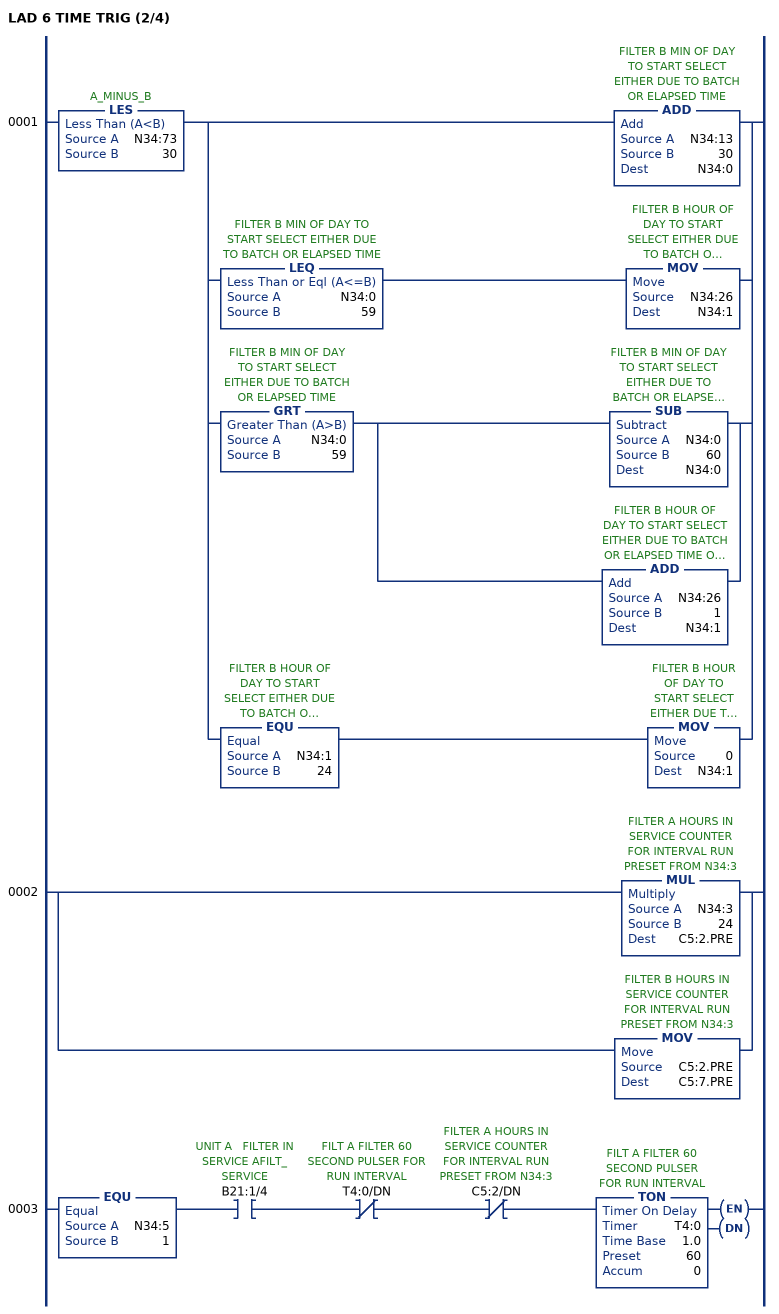
% Rung: 1 %
SOR LES N34:73 30 BST ADD N34:13 30 N34:0 NXB LEQ N34:0 59 MOV N34:26 N34:1 NXB GRT N34:0 59 BST SUB N34:0 60 N34:0 NXB ADD N34:26 1 N34:1 BND NXB EQU N34:1 24 MOV 0 N34:1 BND EOR
%   N34:73  A_MINUS_B %
%   N34:13  "FILTER A MIN OF DAY TO START SELECT EITHER DUE TO BATCH OR ELAPSED TIME" %
%   N34:0  "FILTER B MIN OF DAY TO START SELECT EITHER DUE TO BATCH OR ELAPSED TIME" %
%   N34:26  "FILTER A HOUR OF DAY TO START SELECT EITHER DUE TO BATCH OR ELAPSED TIME OR DP" %
%   N34:1  "FILTER B HOUR OF DAY TO START SELECT EITHER DUE TO BATCH OR ELAPSED TIME OR DP" %
% Rung: 2 %
SOR BST MUL N34:3 24 C5:2.PRE NXB MOV C5:2.PRE C5:7.PRE BND EOR
%   N34:3  "FILT INTERVAL IN DAYS TO START A REGN" %
%   C5:2  "FILTER A HOURS IN SERVICE COUNTER FOR INTERVAL RUN PRESET FROM N34:3" %
%   C5:7  "FILTER B HOURS IN SERVICE COUNTER FOR INTERVAL RUN PRESET FROM N34:3" %
% Rung: 3 %
SOR EQU N34:5 1 XIC B21:1/4 XIO T4:0/DN XIO C5:2/DN TON T4:0 1.0 60 0 EOR
%   B21:1/4  AFILT_SERVICE  "UNIT A   FILTER IN SERVICE" %
%   T4:0  "FILT A FILTER 60 SECOND PULSER FOR RUN INTERVAL" %
%   C5:2  "FILTER A HOURS IN SERVICE COUNTER FOR INTERVAL RUN PRESET FROM N34:3" %

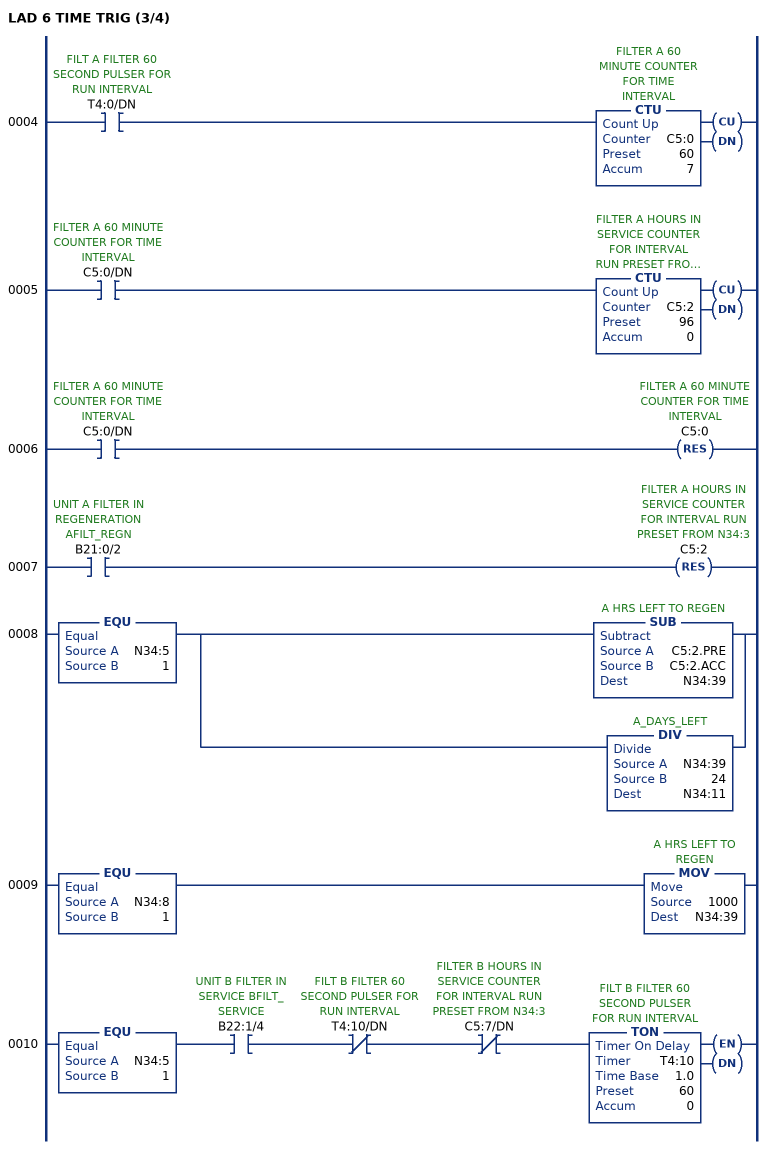
% Rung: 4 %
SOR XIC T4:0/DN CTU C5:0 60 7 EOR
%   T4:0  "FILT A FILTER 60 SECOND PULSER FOR RUN INTERVAL" %
%   C5:0  "FILTER A 60 MINUTE COUNTER FOR TIME INTERVAL" %
% Rung: 5 %
SOR XIC C5:0/DN CTU C5:2 96 0 EOR
%   C5:0  "FILTER A 60 MINUTE COUNTER FOR TIME INTERVAL" %
%   C5:2  "FILTER A HOURS IN SERVICE COUNTER FOR INTERVAL RUN PRESET FROM N34:3" %
% Rung: 6 %
SOR XIC C5:0/DN RES C5:0 EOR
%   C5:0  "FILTER A 60 MINUTE COUNTER FOR TIME INTERVAL" %
% Rung: 7 %
SOR XIC B21:0/2 RES C5:2 EOR
%   B21:0/2  AFILT_REGN  "UNIT A FILTER IN REGENERATION" %
%   C5:2  "FILTER A HOURS IN SERVICE COUNTER FOR INTERVAL RUN PRESET FROM N34:3" %
% Rung: 8 %
SOR EQU N34:5 1 BST SUB C5:2.PRE C5:2.ACC N34:39 NXB DIV N34:39 24 N34:11 BND EOR
%   C5:2  "FILTER A HOURS IN SERVICE COUNTER FOR INTERVAL RUN PRESET FROM N34:3" %
%   N34:39  "A HRS LEFT TO REGEN" %
%   N34:11  A_DAYS_LEFT %
% Rung: 9 %
SOR EQU N34:8 1 MOV 1000 N34:39 EOR
%   N34:39  "A HRS LEFT TO REGEN" %
% Rung: 10 %
SOR EQU N34:5 1 XIC B22:1/4 XIO T4:10/DN XIO C5:7/DN TON T4:10 1.0 60 0 EOR
%   B22:1/4  BFILT_SERVICE  "UNIT B FILTER IN SERVICE" %
%   T4:10  "FILT B FILTER 60 SECOND PULSER FOR RUN INTERVAL" %
%   C5:7  "FILTER B HOURS IN SERVICE COUNTER FOR INTERVAL RUN PRESET FROM N34:3" %

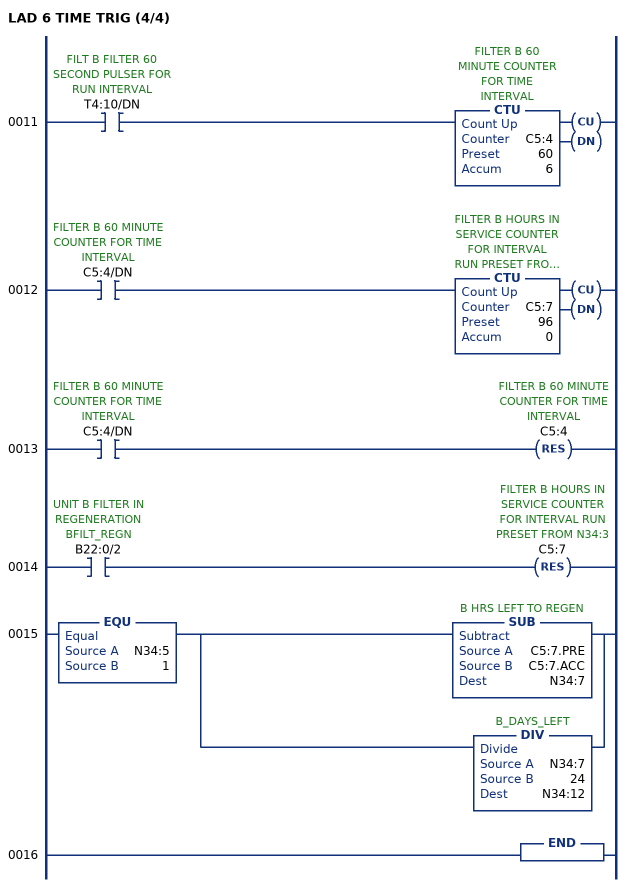
% Rung: 11 %
SOR XIC T4:10/DN CTU C5:4 60 6 EOR
%   T4:10  "FILT B FILTER 60 SECOND PULSER FOR RUN INTERVAL" %
%   C5:4  "FILTER B 60 MINUTE COUNTER FOR TIME INTERVAL" %
% Rung: 12 %
SOR XIC C5:4/DN CTU C5:7 96 0 EOR
%   C5:4  "FILTER B 60 MINUTE COUNTER FOR TIME INTERVAL" %
%   C5:7  "FILTER B HOURS IN SERVICE COUNTER FOR INTERVAL RUN PRESET FROM N34:3" %
% Rung: 13 %
SOR XIC C5:4/DN RES C5:4 EOR
%   C5:4  "FILTER B 60 MINUTE COUNTER FOR TIME INTERVAL" %
% Rung: 14 %
SOR XIC B22:0/2 RES C5:7 EOR
%   B22:0/2  BFILT_REGN  "UNIT B FILTER IN REGENERATION" %
%   C5:7  "FILTER B HOURS IN SERVICE COUNTER FOR INTERVAL RUN PRESET FROM N34:3" %
% Rung: 15 %
SOR EQU N34:5 1 BST SUB C5:7.PRE C5:7.ACC N34:7 NXB DIV N34:7 24 N34:12 BND EOR
%   C5:7  "FILTER B HOURS IN SERVICE COUNTER FOR INTERVAL RUN PRESET FROM N34:3" %
%   N34:7  "B HRS LEFT TO REGEN" %
%   N34:12  B_DAYS_LEFT %
% Rung: 16 %
SOR END EOR

LADDER 7 "A VESSEL"
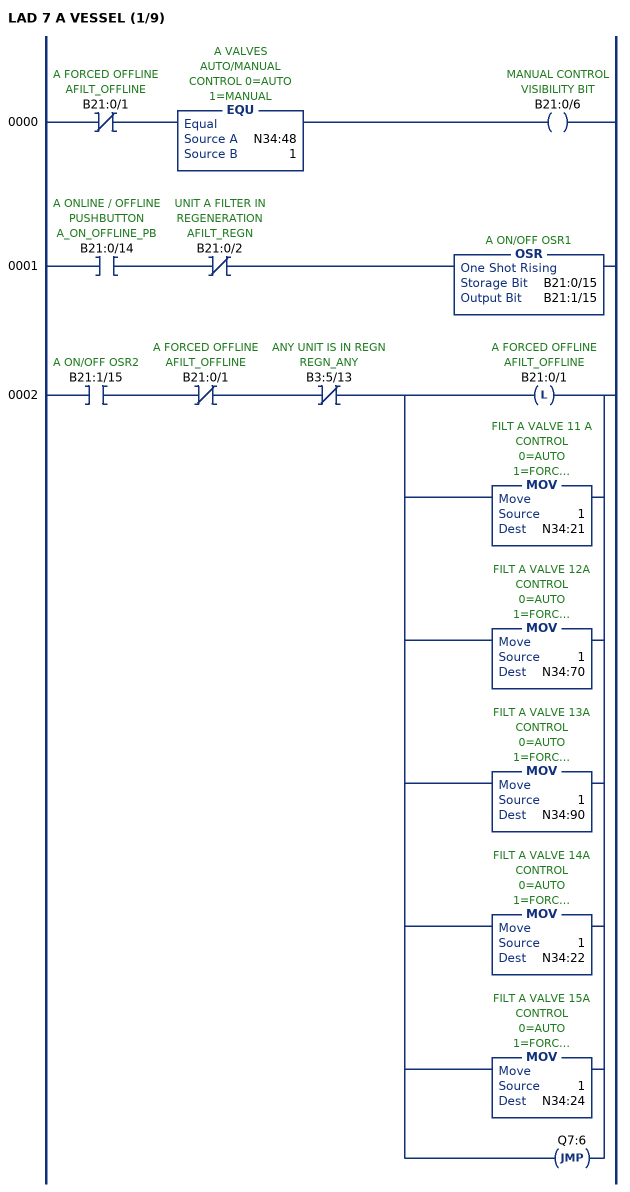
% Rung: 0 %
SOR XIO B21:0/1 EQU N34:48 1 OTE B21:0/6 EOR
%   B21:0/1  AFILT_OFFLINE  "A FORCED OFFLINE" %
%   N34:48  "A VALVES AUTO/MANUAL CONTROL 0=AUTO 1=MANUAL" %
%   B21:0/6  "MANUAL CONTROL VISIBILITY BIT" %
% Rung: 1 %
SOR XIC B21:0/14 XIO B21:0/2 OSR B21:0/15 B21:1/15 EOR
%   B21:0/14  A_ON_OFFLINE_PB  "A ONLINE / OFFLINE PUSHBUTTON" %
%   B21:0/2  AFILT_REGN  "UNIT A FILTER IN REGENERATION" %
%   B21:0/15  "A ON/OFF OSR1" %
%   B21:1/15  "A ON/OFF OSR2" %
% Rung: 2 %
SOR XIC B21:1/15 XIO B21:0/1 XIO B3:5/13 BST OTL B21:0/1 NXB MOV 1 N34:21 NXB MOV 1 N34:70 NXB MOV 1 N34:90 NXB MOV 1 N34:22 NXB MOV 1 N34:24 NXB JMP Q7:6 BND EOR
%   B21:1/15  "A ON/OFF OSR2" %
%   B21:0/1  AFILT_OFFLINE  "A FORCED OFFLINE" %
%   B3:5/13  REGN_ANY  "ANY UNIT IS IN REGN" %
%   N34:21  "FILT A VALVE 11 A CONTROL 0=AUTO 1=FORCE CLOSED 2=FORCE ON" %
%   N34:70  "FILT A VALVE 12A CONTROL 0=AUTO 1=FORCE CLOSED 2=FORCE ON" %
%   N34:90  "FILT A VALVE 13A CONTROL 0=AUTO 1=FORCE CLOSED 2=FORCE ON" %
%   N34:22  "FILT A VALVE 14A CONTROL 0=AUTO 1=FORCE CLOSED 2=FORCE ON" %
%   N34:24  "FILT A VALVE 15A CONTROL 0=AUTO 1=FORCE CLOSED 2=FORCE ON" %

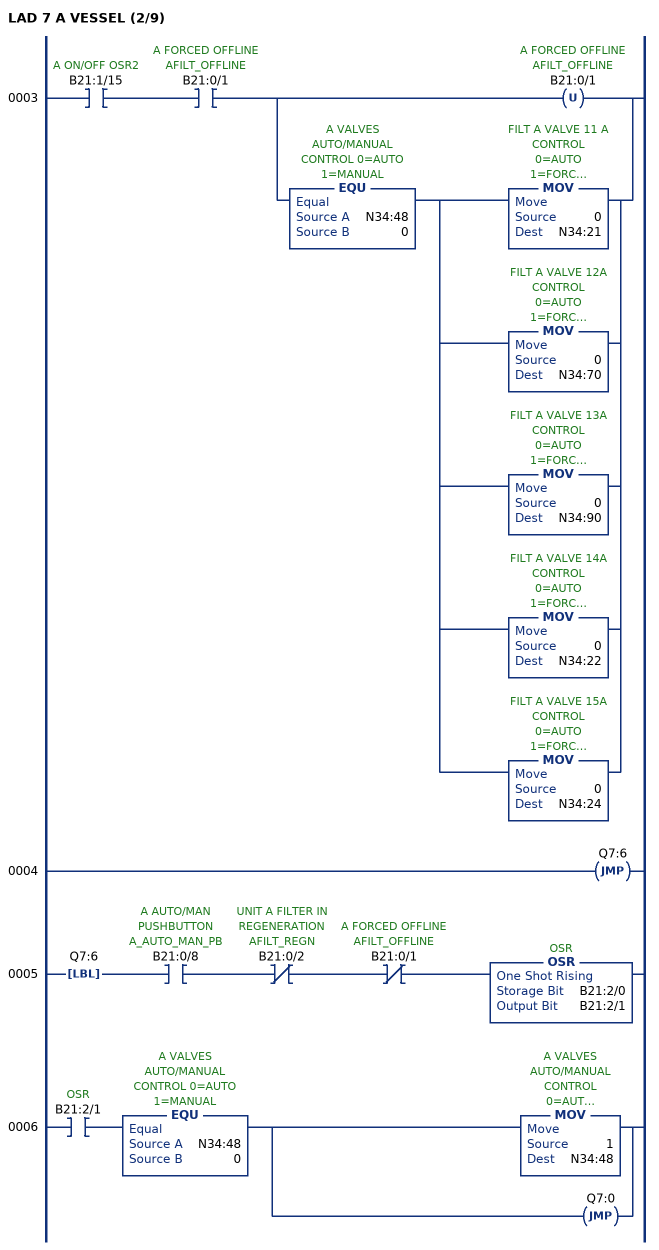
% Rung: 3 %
SOR XIC B21:1/15 XIC B21:0/1 BST OTU B21:0/1 NXB EQU N34:48 0 BST MOV 0 N34:21 NXB MOV 0 N34:70 NXB MOV 0 N34:90 NXB MOV 0 N34:22 NXB MOV 0 N34:24 BND BND EOR
%   B21:1/15  "A ON/OFF OSR2" %
%   B21:0/1  AFILT_OFFLINE  "A FORCED OFFLINE" %
%   N34:48  "A VALVES AUTO/MANUAL CONTROL 0=AUTO 1=MANUAL" %
%   N34:21  "FILT A VALVE 11 A CONTROL 0=AUTO 1=FORCE CLOSED 2=FORCE ON" %
%   N34:70  "FILT A VALVE 12A CONTROL 0=AUTO 1=FORCE CLOSED 2=FORCE ON" %
%   N34:90  "FILT A VALVE 13A CONTROL 0=AUTO 1=FORCE CLOSED 2=FORCE ON" %
%   N34:22  "FILT A VALVE 14A CONTROL 0=AUTO 1=FORCE CLOSED 2=FORCE ON" %
%   N34:24  "FILT A VALVE 15A CONTROL 0=AUTO 1=FORCE CLOSED 2=FORCE ON" %
% Rung: 4 %
SOR JMP Q7:6 EOR
% Rung: 5 %
SOR LBL Q7:6 XIC B21:0/8 XIO B21:0/2 XIO B21:0/1 OSR B21:2/0 B21:2/1 EOR
%   B21:0/8  A_AUTO_MAN_PB  "A AUTO/MAN PUSHBUTTON" %
%   B21:0/2  AFILT_REGN  "UNIT A FILTER IN REGENERATION" %
%   B21:0/1  AFILT_OFFLINE  "A FORCED OFFLINE" %
%   B21:2/0  "OSR" %
%   B21:2/1  "OSR" %
% Rung: 6 %
SOR XIC B21:2/1 EQU N34:48 0 BST MOV 1 N34:48 NXB JMP Q7:0 BND EOR
%   B21:2/1  "OSR" %
%   N34:48  "A VALVES AUTO/MANUAL CONTROL 0=AUTO 1=MANUAL" %

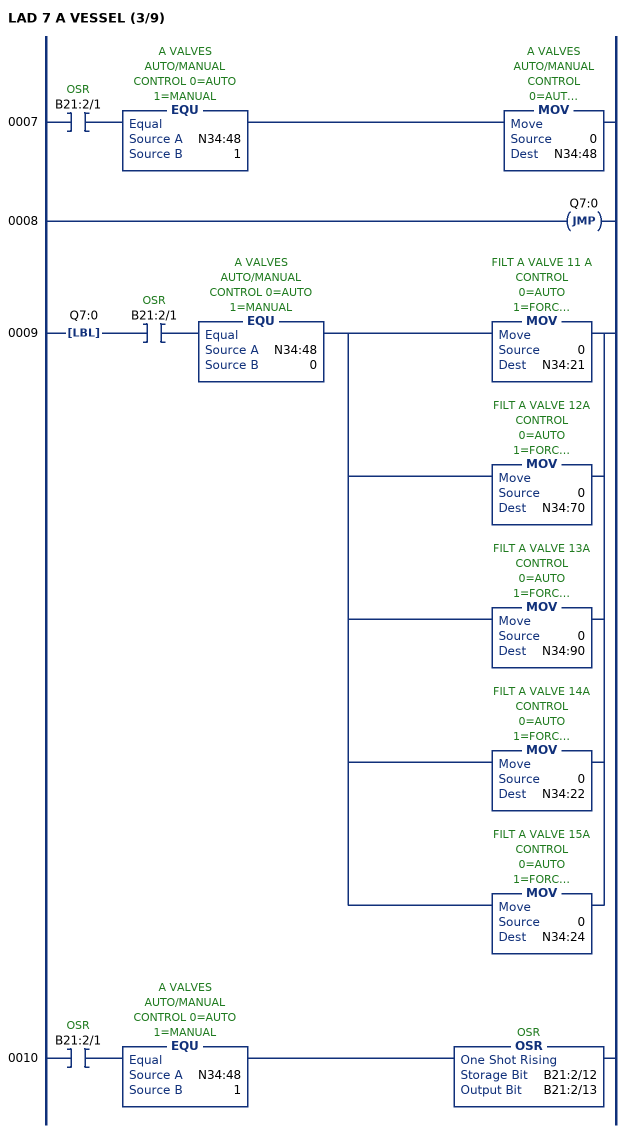
% Rung: 7 %
SOR XIC B21:2/1 EQU N34:48 1 MOV 0 N34:48 EOR
%   B21:2/1  "OSR" %
%   N34:48  "A VALVES AUTO/MANUAL CONTROL 0=AUTO 1=MANUAL" %
% Rung: 8 %
SOR JMP Q7:0 EOR
% Rung: 9 %
SOR LBL Q7:0 XIC B21:2/1 EQU N34:48 0 BST MOV 0 N34:21 NXB MOV 0 N34:70 NXB MOV 0 N34:90 NXB MOV 0 N34:22 NXB MOV 0 N34:24 BND EOR
%   B21:2/1  "OSR" %
%   N34:48  "A VALVES AUTO/MANUAL CONTROL 0=AUTO 1=MANUAL" %
%   N34:21  "FILT A VALVE 11 A CONTROL 0=AUTO 1=FORCE CLOSED 2=FORCE ON" %
%   N34:70  "FILT A VALVE 12A CONTROL 0=AUTO 1=FORCE CLOSED 2=FORCE ON" %
%   N34:90  "FILT A VALVE 13A CONTROL 0=AUTO 1=FORCE CLOSED 2=FORCE ON" %
%   N34:22  "FILT A VALVE 14A CONTROL 0=AUTO 1=FORCE CLOSED 2=FORCE ON" %
%   N34:24  "FILT A VALVE 15A CONTROL 0=AUTO 1=FORCE CLOSED 2=FORCE ON" %
% Rung: 10 %
SOR XIC B21:2/1 EQU N34:48 1 OSR B21:2/12 B21:2/13 EOR
%   B21:2/1  "OSR" %
%   N34:48  "A VALVES AUTO/MANUAL CONTROL 0=AUTO 1=MANUAL" %
%   B21:2/12  "OSR" %
%   B21:2/13  "OSR" %

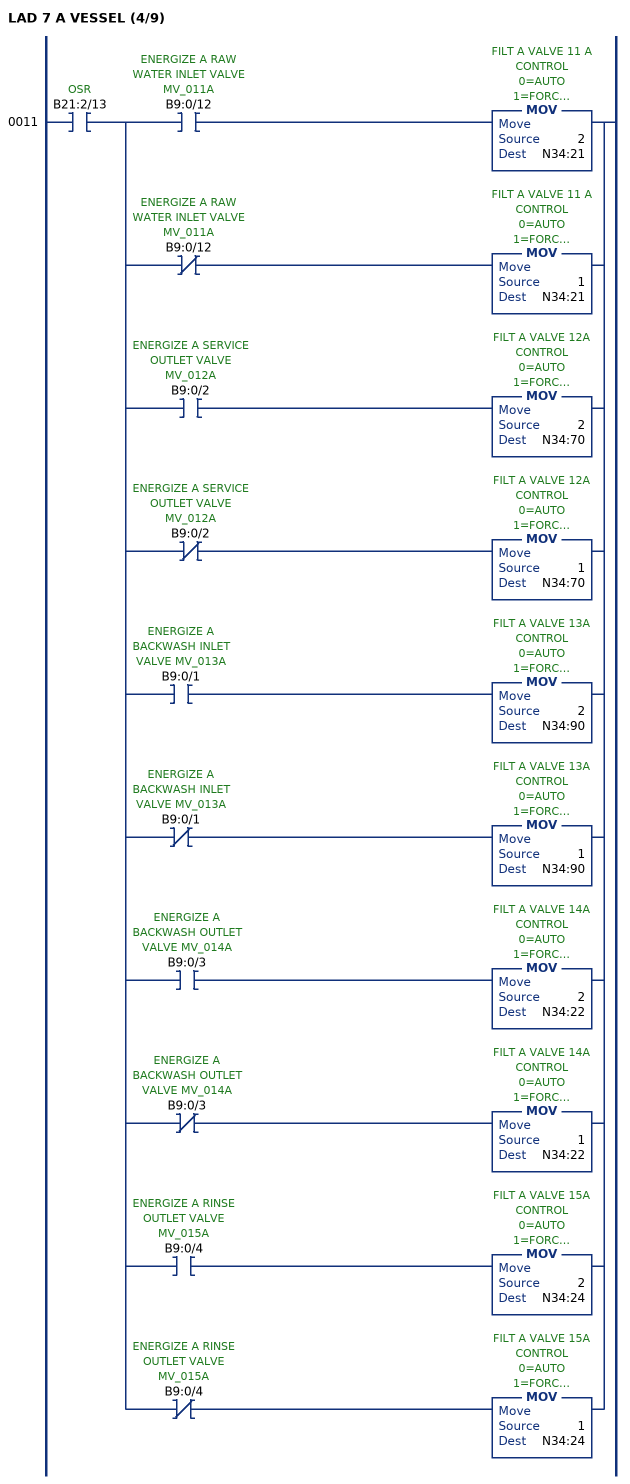
% Rung: 11 %
SOR XIC B21:2/13 BST XIC B9:0/12 MOV 2 N34:21 NXB XIO B9:0/12 MOV 1 N34:21 NXB XIC B9:0/2 MOV 2 N34:70 NXB XIO B9:0/2 MOV 1 N34:70 NXB XIC B9:0/1 MOV 2 N34:90 NXB XIO B9:0/1 MOV 1 N34:90 NXB XIC B9:0/3 MOV 2 N34:22 NXB XIO B9:0/3 MOV 1 N34:22 NXB XIC B9:0/4 MOV 2 N34:24 NXB XIO B9:0/4 MOV 1 N34:24 BND EOR
%   B21:2/13  "OSR" %
%   B9:0/12  MV_011A  "ENERGIZE A RAW WATER INLET VALVE" %
%   N34:21  "FILT A VALVE 11 A CONTROL 0=AUTO 1=FORCE CLOSED 2=FORCE ON" %
%   B9:0/2  MV_012A  "ENERGIZE A SERVICE OUTLET VALVE" %
%   N34:70  "FILT A VALVE 12A CONTROL 0=AUTO 1=FORCE CLOSED 2=FORCE ON" %
%   B9:0/1  MV_013A  "ENERGIZE A BACKWASH INLET VALVE" %
%   N34:90  "FILT A VALVE 13A CONTROL 0=AUTO 1=FORCE CLOSED 2=FORCE ON" %
%   B9:0/3  MV_014A  "ENERGIZE A BACKWASH OUTLET VALVE" %
%   N34:22  "FILT A VALVE 14A CONTROL 0=AUTO 1=FORCE CLOSED 2=FORCE ON" %
%   B9:0/4  MV_015A  "ENERGIZE A RINSE OUTLET VALVE" %
%   N34:24  "FILT A VALVE 15A CONTROL 0=AUTO 1=FORCE CLOSED 2=FORCE ON" %

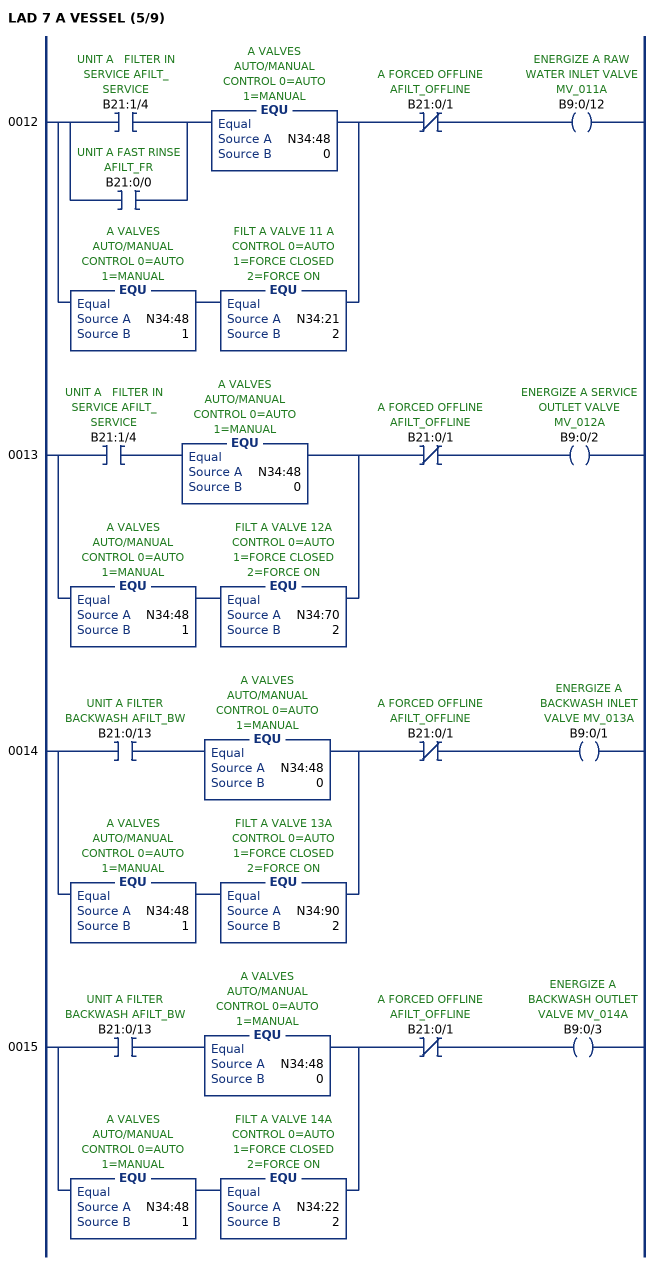
% Rung: 12 %
SOR BST BST XIC B21:1/4 NXB XIC B21:0/0 BND EQU N34:48 0 NXB EQU N34:48 1 EQU N34:21 2 BND XIO B21:0/1 OTE B9:0/12 EOR
%   B21:1/4  AFILT_SERVICE  "UNIT A   FILTER IN SERVICE" %
%   B21:0/0  AFILT_FR  "UNIT A FAST RINSE" %
%   N34:48  "A VALVES AUTO/MANUAL CONTROL 0=AUTO 1=MANUAL" %
%   N34:21  "FILT A VALVE 11 A CONTROL 0=AUTO 1=FORCE CLOSED 2=FORCE ON" %
%   B21:0/1  AFILT_OFFLINE  "A FORCED OFFLINE" %
%   B9:0/12  MV_011A  "ENERGIZE A RAW WATER INLET VALVE" %
% Rung: 13 %
SOR BST XIC B21:1/4 EQU N34:48 0 NXB EQU N34:48 1 EQU N34:70 2 BND XIO B21:0/1 OTE B9:0/2 EOR
%   B21:1/4  AFILT_SERVICE  "UNIT A   FILTER IN SERVICE" %
%   N34:48  "A VALVES AUTO/MANUAL CONTROL 0=AUTO 1=MANUAL" %
%   N34:70  "FILT A VALVE 12A CONTROL 0=AUTO 1=FORCE CLOSED 2=FORCE ON" %
%   B21:0/1  AFILT_OFFLINE  "A FORCED OFFLINE" %
%   B9:0/2  MV_012A  "ENERGIZE A SERVICE OUTLET VALVE" %
% Rung: 14 %
SOR BST XIC B21:0/13 EQU N34:48 0 NXB EQU N34:48 1 EQU N34:90 2 BND XIO B21:0/1 OTE B9:0/1 EOR
%   B21:0/13  AFILT_BW  "UNIT A FILTER BACKWASH" %
%   N34:48  "A VALVES AUTO/MANUAL CONTROL 0=AUTO 1=MANUAL" %
%   N34:90  "FILT A VALVE 13A CONTROL 0=AUTO 1=FORCE CLOSED 2=FORCE ON" %
%   B21:0/1  AFILT_OFFLINE  "A FORCED OFFLINE" %
%   B9:0/1  MV_013A  "ENERGIZE A BACKWASH INLET VALVE" %
% Rung: 15 %
SOR BST XIC B21:0/13 EQU N34:48 0 NXB EQU N34:48 1 EQU N34:22 2 BND XIO B21:0/1 OTE B9:0/3 EOR
%   B21:0/13  AFILT_BW  "UNIT A FILTER BACKWASH" %
%   N34:48  "A VALVES AUTO/MANUAL CONTROL 0=AUTO 1=MANUAL" %
%   N34:22  "FILT A VALVE 14A CONTROL 0=AUTO 1=FORCE CLOSED 2=FORCE ON" %
%   B21:0/1  AFILT_OFFLINE  "A FORCED OFFLINE" %
%   B9:0/3  MV_014A  "ENERGIZE A BACKWASH OUTLET VALVE" %

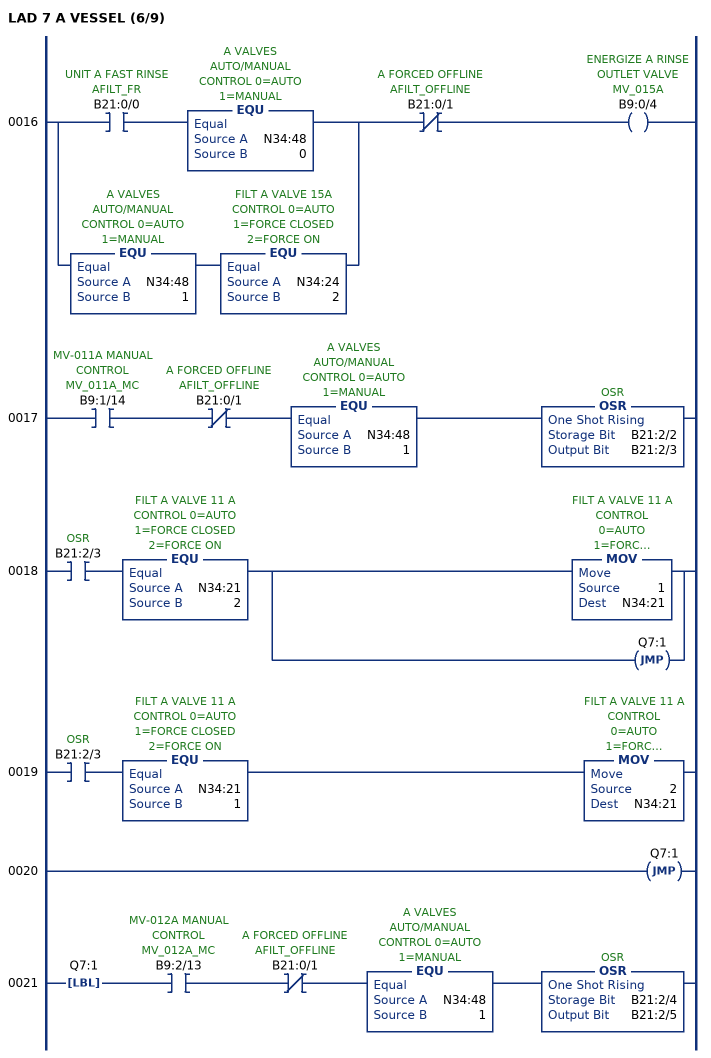
% Rung: 16 %
SOR BST XIC B21:0/0 EQU N34:48 0 NXB EQU N34:48 1 EQU N34:24 2 BND XIO B21:0/1 OTE B9:0/4 EOR
%   B21:0/0  AFILT_FR  "UNIT A FAST RINSE" %
%   N34:48  "A VALVES AUTO/MANUAL CONTROL 0=AUTO 1=MANUAL" %
%   N34:24  "FILT A VALVE 15A CONTROL 0=AUTO 1=FORCE CLOSED 2=FORCE ON" %
%   B21:0/1  AFILT_OFFLINE  "A FORCED OFFLINE" %
%   B9:0/4  MV_015A  "ENERGIZE A RINSE OUTLET VALVE" %
% Rung: 17 %
SOR XIC B9:1/14 XIO B21:0/1 EQU N34:48 1 OSR B21:2/2 B21:2/3 EOR
%   B9:1/14  MV_011A_MC  "MV-011A MANUAL CONTROL" %
%   B21:0/1  AFILT_OFFLINE  "A FORCED OFFLINE" %
%   N34:48  "A VALVES AUTO/MANUAL CONTROL 0=AUTO 1=MANUAL" %
%   B21:2/2  "OSR" %
%   B21:2/3  "OSR" %
% Rung: 18 %
SOR XIC B21:2/3 EQU N34:21 2 BST MOV 1 N34:21 NXB JMP Q7:1 BND EOR
%   B21:2/3  "OSR" %
%   N34:21  "FILT A VALVE 11 A CONTROL 0=AUTO 1=FORCE CLOSED 2=FORCE ON" %
% Rung: 19 %
SOR XIC B21:2/3 EQU N34:21 1 MOV 2 N34:21 EOR
%   B21:2/3  "OSR" %
%   N34:21  "FILT A VALVE 11 A CONTROL 0=AUTO 1=FORCE CLOSED 2=FORCE ON" %
% Rung: 20 %
SOR JMP Q7:1 EOR
% Rung: 21 %
SOR LBL Q7:1 XIC B9:2/13 XIO B21:0/1 EQU N34:48 1 OSR B21:2/4 B21:2/5 EOR
%   B9:2/13  MV_012A_MC  "MV-012A MANUAL CONTROL" %
%   B21:0/1  AFILT_OFFLINE  "A FORCED OFFLINE" %
%   N34:48  "A VALVES AUTO/MANUAL CONTROL 0=AUTO 1=MANUAL" %
%   B21:2/4  "OSR" %
%   B21:2/5  "OSR" %

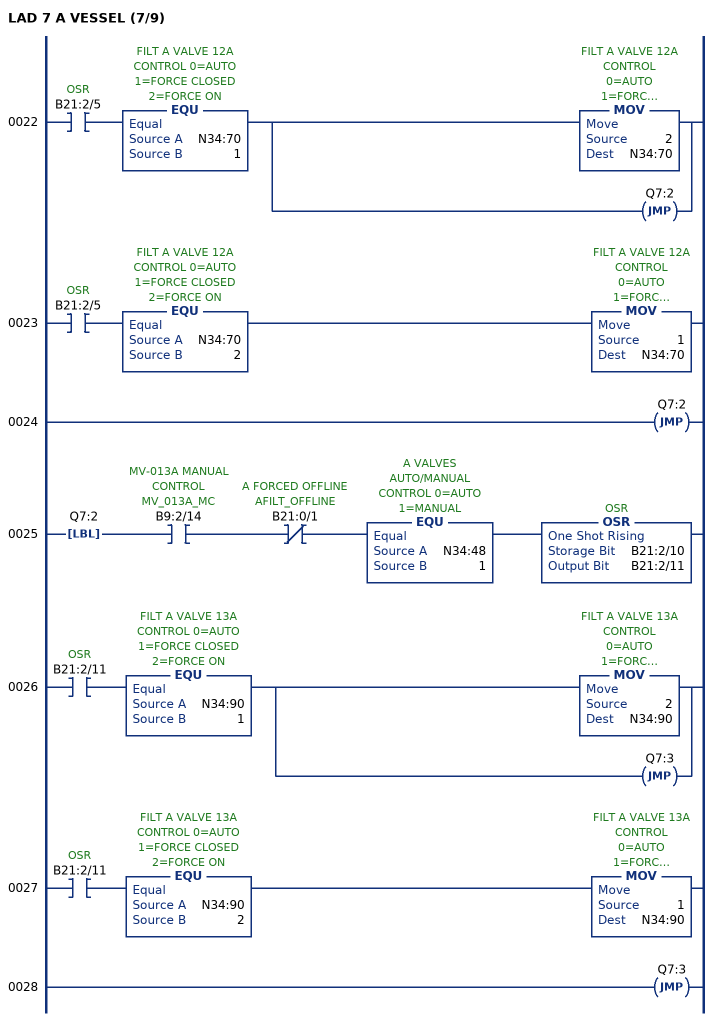
% Rung: 22 %
SOR XIC B21:2/5 EQU N34:70 1 BST MOV 2 N34:70 NXB JMP Q7:2 BND EOR
%   B21:2/5  "OSR" %
%   N34:70  "FILT A VALVE 12A CONTROL 0=AUTO 1=FORCE CLOSED 2=FORCE ON" %
% Rung: 23 %
SOR XIC B21:2/5 EQU N34:70 2 MOV 1 N34:70 EOR
%   B21:2/5  "OSR" %
%   N34:70  "FILT A VALVE 12A CONTROL 0=AUTO 1=FORCE CLOSED 2=FORCE ON" %
% Rung: 24 %
SOR JMP Q7:2 EOR
% Rung: 25 %
SOR LBL Q7:2 XIC B9:2/14 XIO B21:0/1 EQU N34:48 1 OSR B21:2/10 B21:2/11 EOR
%   B9:2/14  MV_013A_MC  "MV-013A MANUAL CONTROL" %
%   B21:0/1  AFILT_OFFLINE  "A FORCED OFFLINE" %
%   N34:48  "A VALVES AUTO/MANUAL CONTROL 0=AUTO 1=MANUAL" %
%   B21:2/10  "OSR" %
%   B21:2/11  "OSR" %
% Rung: 26 %
SOR XIC B21:2/11 EQU N34:90 1 BST MOV 2 N34:90 NXB JMP Q7:3 BND EOR
%   B21:2/11  "OSR" %
%   N34:90  "FILT A VALVE 13A CONTROL 0=AUTO 1=FORCE CLOSED 2=FORCE ON" %
% Rung: 27 %
SOR XIC B21:2/11 EQU N34:90 2 MOV 1 N34:90 EOR
%   B21:2/11  "OSR" %
%   N34:90  "FILT A VALVE 13A CONTROL 0=AUTO 1=FORCE CLOSED 2=FORCE ON" %
% Rung: 28 %
SOR JMP Q7:3 EOR

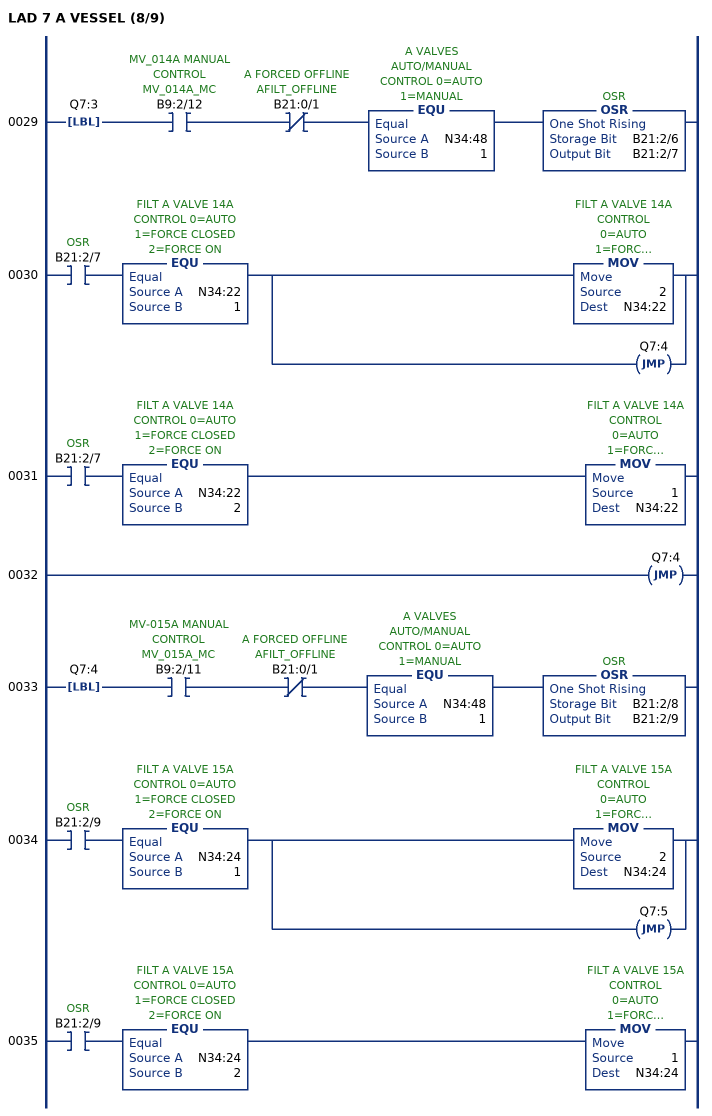
% Rung: 29 %
SOR LBL Q7:3 XIC B9:2/12 XIO B21:0/1 EQU N34:48 1 OSR B21:2/6 B21:2/7 EOR
%   B9:2/12  MV_014A_MC  "MV_014A MANUAL CONTROL" %
%   B21:0/1  AFILT_OFFLINE  "A FORCED OFFLINE" %
%   N34:48  "A VALVES AUTO/MANUAL CONTROL 0=AUTO 1=MANUAL" %
%   B21:2/6  "OSR" %
%   B21:2/7  "OSR" %
% Rung: 30 %
SOR XIC B21:2/7 EQU N34:22 1 BST MOV 2 N34:22 NXB JMP Q7:4 BND EOR
%   B21:2/7  "OSR" %
%   N34:22  "FILT A VALVE 14A CONTROL 0=AUTO 1=FORCE CLOSED 2=FORCE ON" %
% Rung: 31 %
SOR XIC B21:2/7 EQU N34:22 2 MOV 1 N34:22 EOR
%   B21:2/7  "OSR" %
%   N34:22  "FILT A VALVE 14A CONTROL 0=AUTO 1=FORCE CLOSED 2=FORCE ON" %
% Rung: 32 %
SOR JMP Q7:4 EOR
% Rung: 33 %
SOR LBL Q7:4 XIC B9:2/11 XIO B21:0/1 EQU N34:48 1 OSR B21:2/8 B21:2/9 EOR
%   B9:2/11  MV_015A_MC  "MV-015A MANUAL CONTROL" %
%   B21:0/1  AFILT_OFFLINE  "A FORCED OFFLINE" %
%   N34:48  "A VALVES AUTO/MANUAL CONTROL 0=AUTO 1=MANUAL" %
%   B21:2/8  "OSR" %
%   B21:2/9  "OSR" %
% Rung: 34 %
SOR XIC B21:2/9 EQU N34:24 1 BST MOV 2 N34:24 NXB JMP Q7:5 BND EOR
%   B21:2/9  "OSR" %
%   N34:24  "FILT A VALVE 15A CONTROL 0=AUTO 1=FORCE CLOSED 2=FORCE ON" %
% Rung: 35 %
SOR XIC B21:2/9 EQU N34:24 2 MOV 1 N34:24 EOR
%   B21:2/9  "OSR" %
%   N34:24  "FILT A VALVE 15A CONTROL 0=AUTO 1=FORCE CLOSED 2=FORCE ON" %

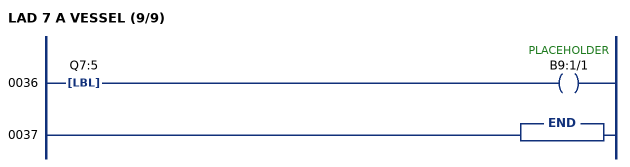
% Rung: 36 %
SOR LBL Q7:5 OTE B9:1/1 EOR
%   B9:1/1  "PLACEHOLDER" %
% Rung: 37 %
SOR END EOR

LADDER 8 "ANALOG IN"
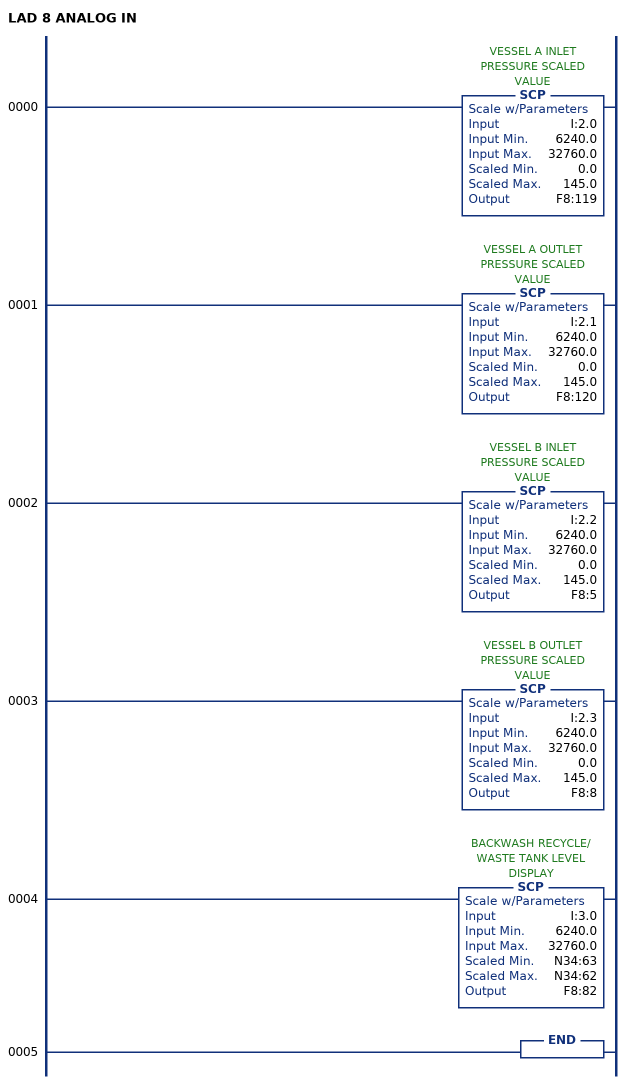
% Rung: 0 %
SOR SCP I:2.0 6240.0 32760.0 0.0 145.0 F8:119 EOR
%   I:2.0  "VESSEL A INLET PRESSURE SCALED VALUE" %
%   F8:119  "VESSEL A INLET PRESSURE SCALED VALUE" %
% Rung: 1 %
SOR SCP I:2.1 6240.0 32760.0 0.0 145.0 F8:120 EOR
%   I:2.1  "VESSEL A OUTLET PRESSURE SCALED VALUE" %
%   F8:120  "VESSEL A OUTLET PRESSURE SCALED VALUE" %
% Rung: 2 %
SOR SCP I:2.2 6240.0 32760.0 0.0 145.0 F8:5 EOR
%   I:2.2  "VESSEL B INLET PRESSURE SCALED VALUE" %
%   F8:5  "VESSEL B INLET PRESSURE SCALED VALUE" %
% Rung: 3 %
SOR SCP I:2.3 6240.0 32760.0 0.0 145.0 F8:8 EOR
%   I:2.3  "VESSEL B OUTLET PRESSURE SCALED VALUE" %
%   F8:8  "VESSEL B OUTLET PRESSURE SCALED VALUE" %
% Rung: 4 %
SOR SCP I:3.0 6240.0 32760.0 N34:63 N34:62 F8:82 EOR
%   I:3.0  "RECYCLE TANK LEVEL TRANSMITTER 4-20" %
%   N34:63  "TANK LO SCALE" %
%   N34:62  "TANK HI SCALE" %
%   F8:82  "BACKWASH RECYCLE/WASTE TANK LEVEL DISPLAY" %
% Rung: 5 %
SOR END EOR

LADDER 9 "PRESSURE"
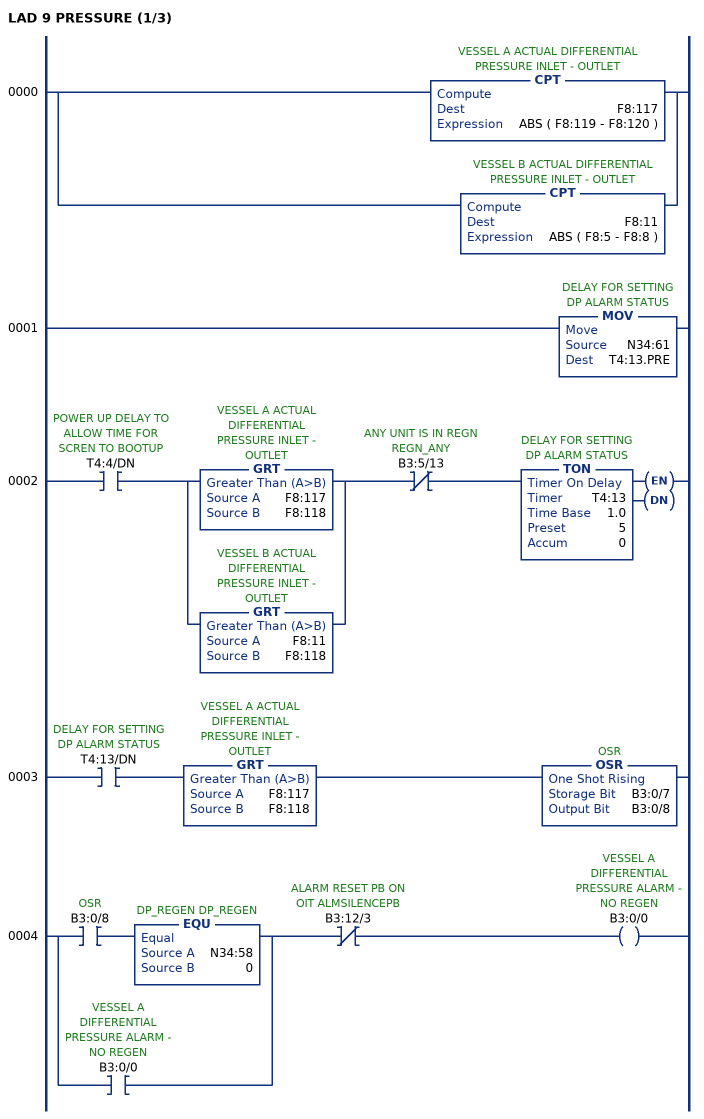
% Rung: 0 %
SOR BST CPT F8:117 " ABS ( F8:119 - F8:120 ) " NXB CPT F8:11 " ABS ( F8:5 - F8:8 ) " BND EOR
%   F8:117  "VESSEL A ACTUAL DIFFERENTIAL PRESSURE INLET - OUTLET" %
%   F8:119  "VESSEL A INLET PRESSURE SCALED VALUE" %
%   F8:120  "VESSEL A OUTLET PRESSURE SCALED VALUE" %
%   F8:11  "VESSEL B ACTUAL DIFFERENTIAL PRESSURE INLET - OUTLET" %
%   F8:5  "VESSEL B INLET PRESSURE SCALED VALUE" %
%   F8:8  "VESSEL B OUTLET PRESSURE SCALED VALUE" %
% Rung: 1 %
SOR MOV N34:61 T4:13.PRE EOR
%   N34:61  "DP DELAY IN SECS FROM HMI" %
%   T4:13  "DELAY FOR SETTING DP ALARM STATUS" %
% Rung: 2 %
SOR XIC T4:4/DN BST GRT F8:117 F8:118 NXB GRT F8:11 F8:118 BND XIO B3:5/13 TON T4:13 1.0 5 0 EOR
%   T4:4  "POWER UP DELAY TO ALLOW TIME FOR SCREN TO BOOTUP" %
%   F8:117  "VESSEL A ACTUAL DIFFERENTIAL PRESSURE INLET - OUTLET" %
%   F8:118  DP_SETPOINT  "PRESSURE DIFFERENTIAL SETPOINT" %
%   F8:11  "VESSEL B ACTUAL DIFFERENTIAL PRESSURE INLET - OUTLET" %
%   B3:5/13  REGN_ANY  "ANY UNIT IS IN REGN" %
%   T4:13  "DELAY FOR SETTING DP ALARM STATUS" %
% Rung: 3 %
SOR XIC T4:13/DN GRT F8:117 F8:118 OSR B3:0/7 B3:0/8 EOR
%   T4:13  "DELAY FOR SETTING DP ALARM STATUS" %
%   F8:117  "VESSEL A ACTUAL DIFFERENTIAL PRESSURE INLET - OUTLET" %
%   F8:118  DP_SETPOINT  "PRESSURE DIFFERENTIAL SETPOINT" %
%   B3:0/7  "OSR" %
%   B3:0/8  "OSR" %
% Rung: 4 %
SOR BST XIC B3:0/8 EQU N34:58 0 NXB XIC B3:0/0 BND XIO B3:12/3 OTE B3:0/0 EOR
%   B3:0/8  "OSR" %
%   N34:58  DP_REGEN  "DP_REGEN" %
%   B3:0/0  "VESSEL A DIFFERENTIAL PRESSURE ALARM - NO REGEN" %
%   B3:12/3  ALMSILENCEPB  "ALARM RESET PB ON OIT" %

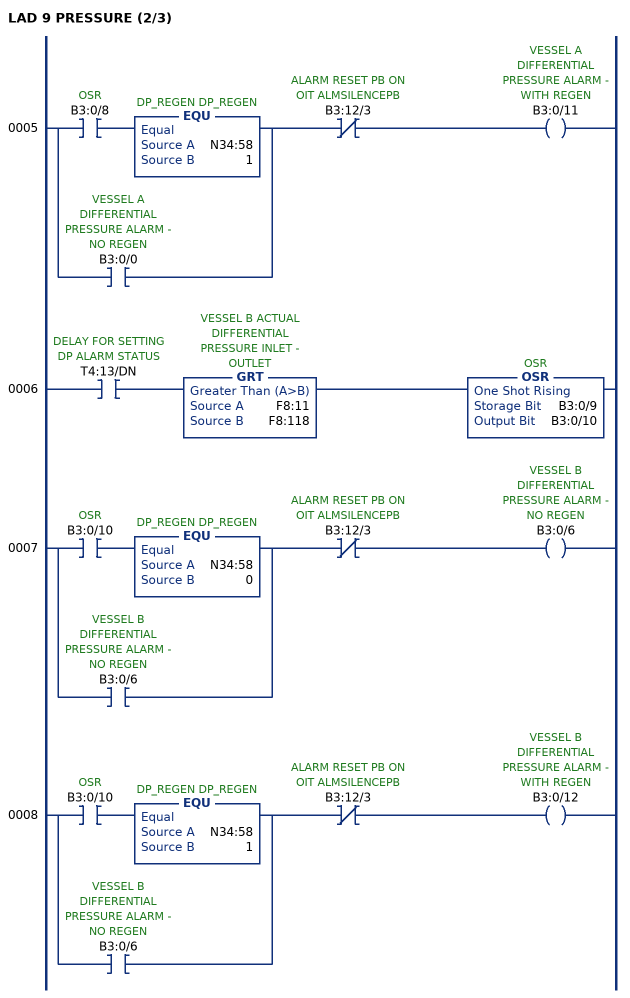
% Rung: 5 %
SOR BST XIC B3:0/8 EQU N34:58 1 NXB XIC B3:0/0 BND XIO B3:12/3 OTE B3:0/11 EOR
%   B3:0/8  "OSR" %
%   N34:58  DP_REGEN  "DP_REGEN" %
%   B3:0/0  "VESSEL A DIFFERENTIAL PRESSURE ALARM - NO REGEN" %
%   B3:12/3  ALMSILENCEPB  "ALARM RESET PB ON OIT" %
%   B3:0/11  "VESSEL A DIFFERENTIAL PRESSURE ALARM - WITH REGEN" %
% Rung: 6 %
SOR XIC T4:13/DN GRT F8:11 F8:118 OSR B3:0/9 B3:0/10 EOR
%   T4:13  "DELAY FOR SETTING DP ALARM STATUS" %
%   F8:11  "VESSEL B ACTUAL DIFFERENTIAL PRESSURE INLET - OUTLET" %
%   F8:118  DP_SETPOINT  "PRESSURE DIFFERENTIAL SETPOINT" %
%   B3:0/9  "OSR" %
%   B3:0/10  "OSR" %
% Rung: 7 %
SOR BST XIC B3:0/10 EQU N34:58 0 NXB XIC B3:0/6 BND XIO B3:12/3 OTE B3:0/6 EOR
%   B3:0/10  "OSR" %
%   N34:58  DP_REGEN  "DP_REGEN" %
%   B3:0/6  "VESSEL B DIFFERENTIAL PRESSURE ALARM - NO REGEN" %
%   B3:12/3  ALMSILENCEPB  "ALARM RESET PB ON OIT" %
% Rung: 8 %
SOR BST XIC B3:0/10 EQU N34:58 1 NXB XIC B3:0/6 BND XIO B3:12/3 OTE B3:0/12 EOR
%   B3:0/10  "OSR" %
%   N34:58  DP_REGEN  "DP_REGEN" %
%   B3:0/6  "VESSEL B DIFFERENTIAL PRESSURE ALARM - NO REGEN" %
%   B3:12/3  ALMSILENCEPB  "ALARM RESET PB ON OIT" %
%   B3:0/12  "VESSEL B DIFFERENTIAL PRESSURE ALARM - WITH REGEN" %

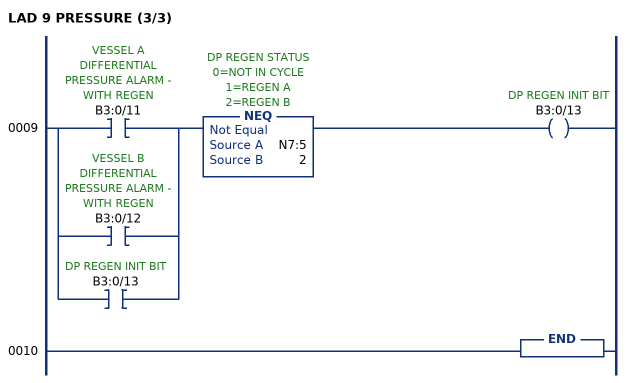
% Rung: 9 %
SOR BST XIC B3:0/11 NXB XIC B3:0/12 NXB XIC B3:0/13 BND NEQ N7:5 2 OTE B3:0/13 EOR
%   B3:0/11  "VESSEL A DIFFERENTIAL PRESSURE ALARM - WITH REGEN" %
%   B3:0/12  "VESSEL B DIFFERENTIAL PRESSURE ALARM - WITH REGEN" %
%   B3:0/13  "DP REGEN INIT BIT" %
%   N7:5  "DP REGEN STATUS 0=NOT IN CYCLE 1=REGEN A 2=REGEN B" %
% Rung: 10 %
SOR END EOR

LADDER 10 "B VESSEL"
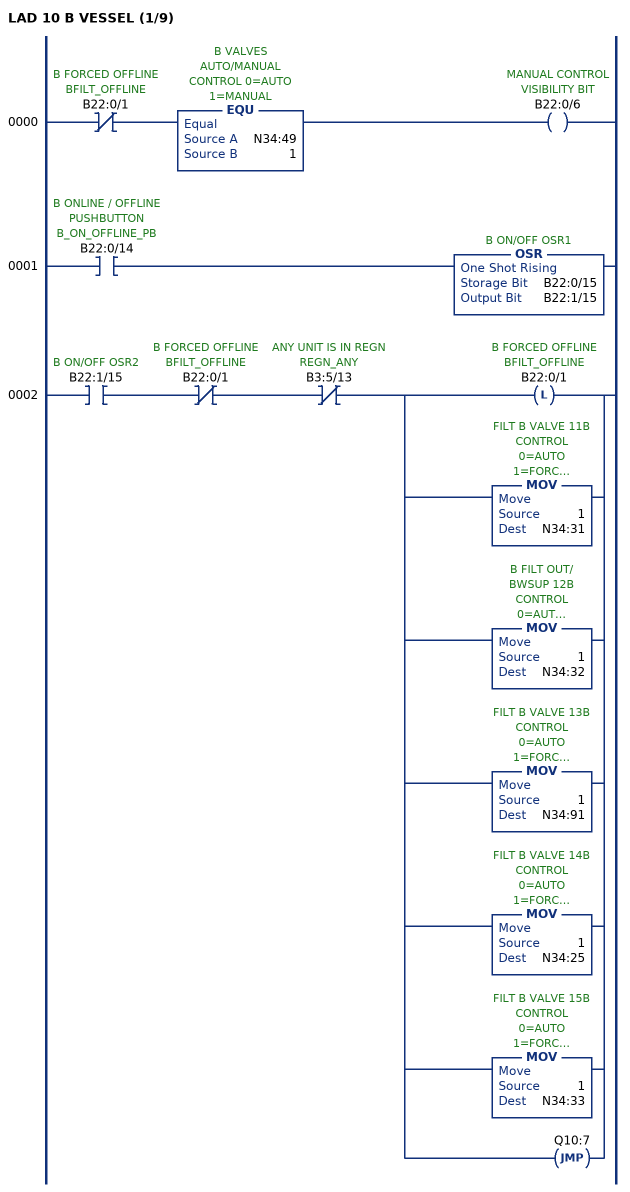
% Rung: 0 %
SOR XIO B22:0/1 EQU N34:49 1 OTE B22:0/6 EOR
%   B22:0/1  BFILT_OFFLINE  "B FORCED OFFLINE" %
%   N34:49  "B VALVES AUTO/MANUAL CONTROL 0=AUTO 1=MANUAL" %
%   B22:0/6  "MANUAL CONTROL VISIBILITY BIT" %
% Rung: 1 %
SOR XIC B22:0/14 OSR B22:0/15 B22:1/15 EOR
%   B22:0/14  B_ON_OFFLINE_PB  "B ONLINE / OFFLINE PUSHBUTTON" %
%   B22:0/15  "B ON/OFF OSR1" %
%   B22:1/15  "B ON/OFF OSR2" %
% Rung: 2 %
SOR XIC B22:1/15 XIO B22:0/1 XIO B3:5/13 BST OTL B22:0/1 NXB MOV 1 N34:31 NXB MOV 1 N34:32 NXB MOV 1 N34:91 NXB MOV 1 N34:25 NXB MOV 1 N34:33 NXB JMP Q10:7 BND EOR
%   B22:1/15  "B ON/OFF OSR2" %
%   B22:0/1  BFILT_OFFLINE  "B FORCED OFFLINE" %
%   B3:5/13  REGN_ANY  "ANY UNIT IS IN REGN" %
%   N34:31  "FILT B VALVE 11B CONTROL 0=AUTO 1=FORCE CLOSED 2=FORCE ON" %
%   N34:32  "B FILT OUT/BWSUP 12B CONTROL 0=AUTO 1=FORCE CLOSED 2=FORCE ON" %
%   N34:91  "FILT B VALVE 13B CONTROL 0=AUTO 1=FORCE CLOSED 2=FORCE ON" %
%   N34:25  "FILT B VALVE 14B CONTROL 0=AUTO 1=FORCE CLOSED 2=FORCE ON" %
%   N34:33  "FILT B VALVE 15B CONTROL 0=AUTO 1=FORCE CLOSED 2=FORCE ON" %

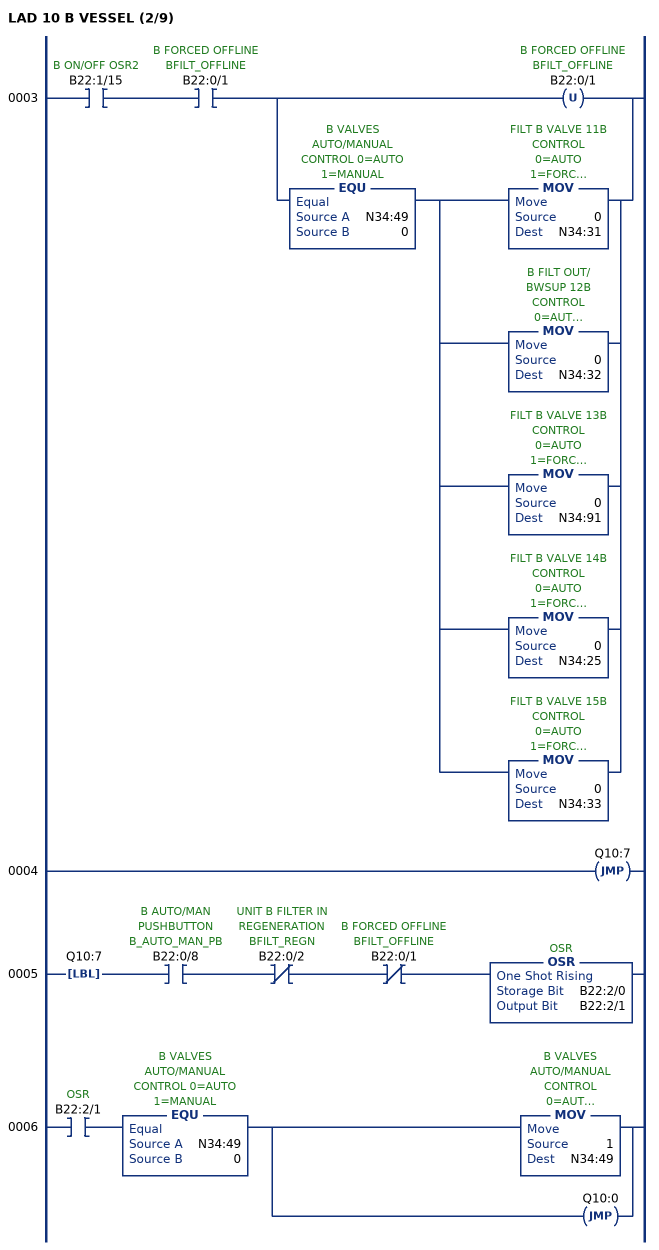
% Rung: 3 %
SOR XIC B22:1/15 XIC B22:0/1 BST OTU B22:0/1 NXB EQU N34:49 0 BST MOV 0 N34:31 NXB MOV 0 N34:32 NXB MOV 0 N34:91 NXB MOV 0 N34:25 NXB MOV 0 N34:33 BND BND EOR
%   B22:1/15  "B ON/OFF OSR2" %
%   B22:0/1  BFILT_OFFLINE  "B FORCED OFFLINE" %
%   N34:49  "B VALVES AUTO/MANUAL CONTROL 0=AUTO 1=MANUAL" %
%   N34:31  "FILT B VALVE 11B CONTROL 0=AUTO 1=FORCE CLOSED 2=FORCE ON" %
%   N34:32  "B FILT OUT/BWSUP 12B CONTROL 0=AUTO 1=FORCE CLOSED 2=FORCE ON" %
%   N34:91  "FILT B VALVE 13B CONTROL 0=AUTO 1=FORCE CLOSED 2=FORCE ON" %
%   N34:25  "FILT B VALVE 14B CONTROL 0=AUTO 1=FORCE CLOSED 2=FORCE ON" %
%   N34:33  "FILT B VALVE 15B CONTROL 0=AUTO 1=FORCE CLOSED 2=FORCE ON" %
% Rung: 4 %
SOR JMP Q10:7 EOR
% Rung: 5 %
SOR LBL Q10:7 XIC B22:0/8 XIO B22:0/2 XIO B22:0/1 OSR B22:2/0 B22:2/1 EOR
%   B22:0/8  B_AUTO_MAN_PB  "B AUTO/MAN PUSHBUTTON" %
%   B22:0/2  BFILT_REGN  "UNIT B FILTER IN REGENERATION" %
%   B22:0/1  BFILT_OFFLINE  "B FORCED OFFLINE" %
%   B22:2/0  "OSR" %
%   B22:2/1  "OSR" %
% Rung: 6 %
SOR XIC B22:2/1 EQU N34:49 0 BST MOV 1 N34:49 NXB JMP Q10:0 BND EOR
%   B22:2/1  "OSR" %
%   N34:49  "B VALVES AUTO/MANUAL CONTROL 0=AUTO 1=MANUAL" %

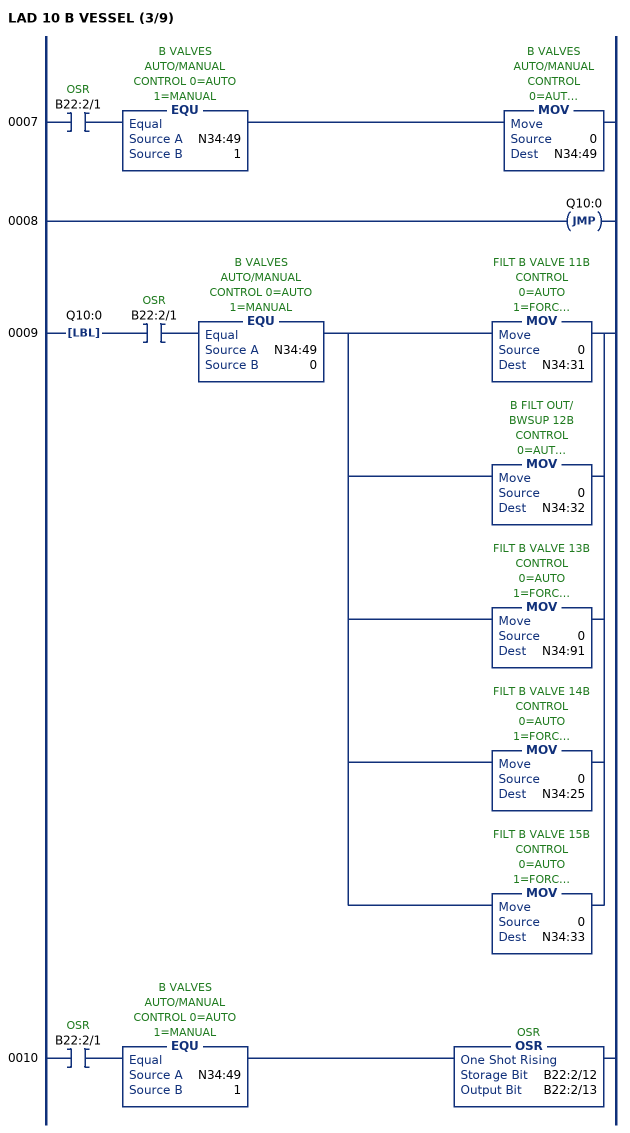
% Rung: 7 %
SOR XIC B22:2/1 EQU N34:49 1 MOV 0 N34:49 EOR
%   B22:2/1  "OSR" %
%   N34:49  "B VALVES AUTO/MANUAL CONTROL 0=AUTO 1=MANUAL" %
% Rung: 8 %
SOR JMP Q10:0 EOR
% Rung: 9 %
SOR LBL Q10:0 XIC B22:2/1 EQU N34:49 0 BST MOV 0 N34:31 NXB MOV 0 N34:32 NXB MOV 0 N34:91 NXB MOV 0 N34:25 NXB MOV 0 N34:33 BND EOR
%   B22:2/1  "OSR" %
%   N34:49  "B VALVES AUTO/MANUAL CONTROL 0=AUTO 1=MANUAL" %
%   N34:31  "FILT B VALVE 11B CONTROL 0=AUTO 1=FORCE CLOSED 2=FORCE ON" %
%   N34:32  "B FILT OUT/BWSUP 12B CONTROL 0=AUTO 1=FORCE CLOSED 2=FORCE ON" %
%   N34:91  "FILT B VALVE 13B CONTROL 0=AUTO 1=FORCE CLOSED 2=FORCE ON" %
%   N34:25  "FILT B VALVE 14B CONTROL 0=AUTO 1=FORCE CLOSED 2=FORCE ON" %
%   N34:33  "FILT B VALVE 15B CONTROL 0=AUTO 1=FORCE CLOSED 2=FORCE ON" %
% Rung: 10 %
SOR XIC B22:2/1 EQU N34:49 1 OSR B22:2/12 B22:2/13 EOR
%   B22:2/1  "OSR" %
%   N34:49  "B VALVES AUTO/MANUAL CONTROL 0=AUTO 1=MANUAL" %
%   B22:2/12  "OSR" %
%   B22:2/13  "OSR" %

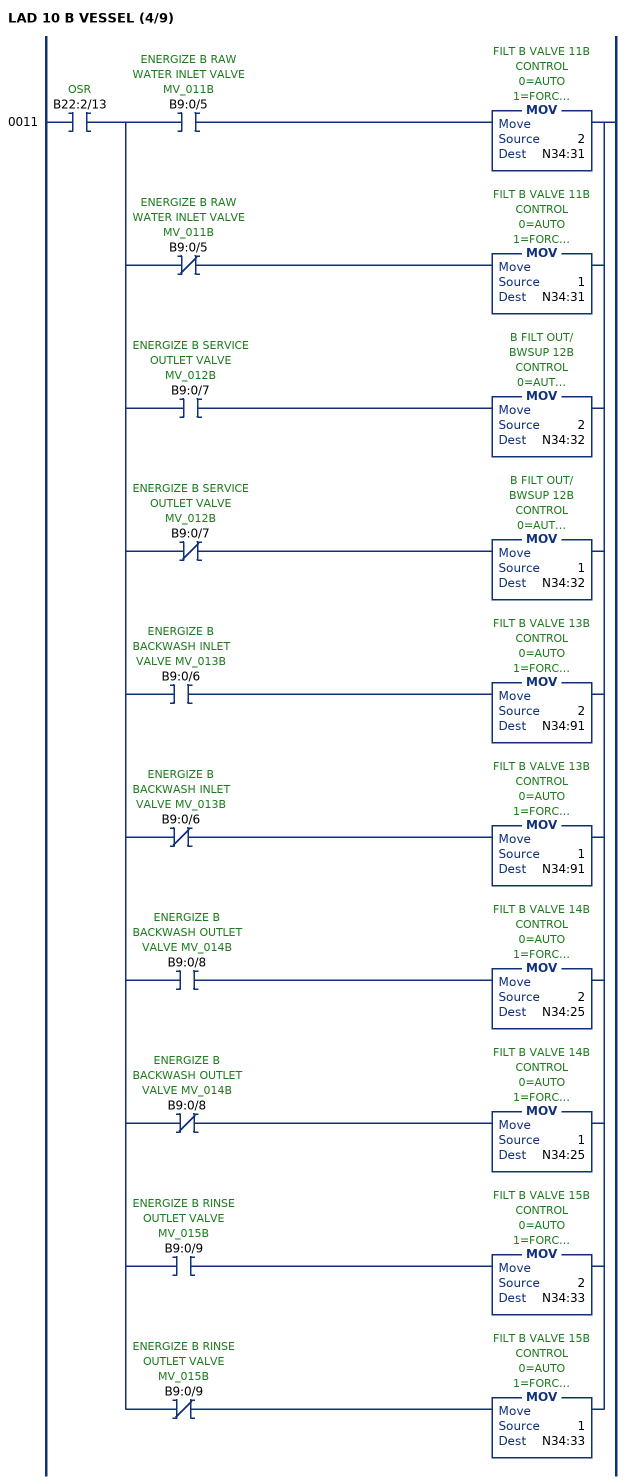
% Rung: 11 %
SOR XIC B22:2/13 BST XIC B9:0/5 MOV 2 N34:31 NXB XIO B9:0/5 MOV 1 N34:31 NXB XIC B9:0/7 MOV 2 N34:32 NXB XIO B9:0/7 MOV 1 N34:32 NXB XIC B9:0/6 MOV 2 N34:91 NXB XIO B9:0/6 MOV 1 N34:91 NXB XIC B9:0/8 MOV 2 N34:25 NXB XIO B9:0/8 MOV 1 N34:25 NXB XIC B9:0/9 MOV 2 N34:33 NXB XIO B9:0/9 MOV 1 N34:33 BND EOR
%   B22:2/13  "OSR" %
%   B9:0/5  MV_011B  "ENERGIZE B RAW WATER INLET VALVE" %
%   N34:31  "FILT B VALVE 11B CONTROL 0=AUTO 1=FORCE CLOSED 2=FORCE ON" %
%   B9:0/7  MV_012B  "ENERGIZE B SERVICE OUTLET VALVE" %
%   N34:32  "B FILT OUT/BWSUP 12B CONTROL 0=AUTO 1=FORCE CLOSED 2=FORCE ON" %
%   B9:0/6  MV_013B  "ENERGIZE B BACKWASH INLET VALVE" %
%   N34:91  "FILT B VALVE 13B CONTROL 0=AUTO 1=FORCE CLOSED 2=FORCE ON" %
%   B9:0/8  MV_014B  "ENERGIZE B BACKWASH OUTLET VALVE" %
%   N34:25  "FILT B VALVE 14B CONTROL 0=AUTO 1=FORCE CLOSED 2=FORCE ON" %
%   B9:0/9  MV_015B  "ENERGIZE B RINSE OUTLET VALVE" %
%   N34:33  "FILT B VALVE 15B CONTROL 0=AUTO 1=FORCE CLOSED 2=FORCE ON" %

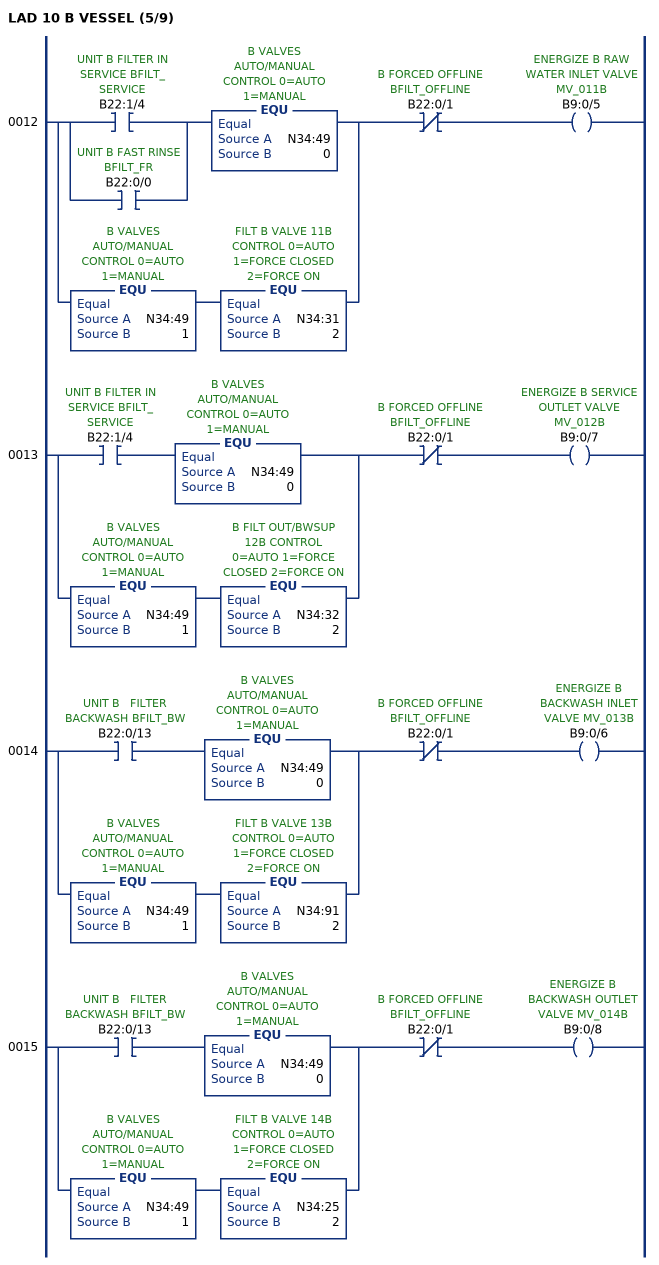
% Rung: 12 %
SOR BST BST XIC B22:1/4 NXB XIC B22:0/0 BND EQU N34:49 0 NXB EQU N34:49 1 EQU N34:31 2 BND XIO B22:0/1 OTE B9:0/5 EOR
%   B22:1/4  BFILT_SERVICE  "UNIT B FILTER IN SERVICE" %
%   B22:0/0  BFILT_FR  "UNIT B FAST RINSE" %
%   N34:49  "B VALVES AUTO/MANUAL CONTROL 0=AUTO 1=MANUAL" %
%   N34:31  "FILT B VALVE 11B CONTROL 0=AUTO 1=FORCE CLOSED 2=FORCE ON" %
%   B22:0/1  BFILT_OFFLINE  "B FORCED OFFLINE" %
%   B9:0/5  MV_011B  "ENERGIZE B RAW WATER INLET VALVE" %
% Rung: 13 %
SOR BST XIC B22:1/4 EQU N34:49 0 NXB EQU N34:49 1 EQU N34:32 2 BND XIO B22:0/1 OTE B9:0/7 EOR
%   B22:1/4  BFILT_SERVICE  "UNIT B FILTER IN SERVICE" %
%   N34:49  "B VALVES AUTO/MANUAL CONTROL 0=AUTO 1=MANUAL" %
%   N34:32  "B FILT OUT/BWSUP 12B CONTROL 0=AUTO 1=FORCE CLOSED 2=FORCE ON" %
%   B22:0/1  BFILT_OFFLINE  "B FORCED OFFLINE" %
%   B9:0/7  MV_012B  "ENERGIZE B SERVICE OUTLET VALVE" %
% Rung: 14 %
SOR BST XIC B22:0/13 EQU N34:49 0 NXB EQU N34:49 1 EQU N34:91 2 BND XIO B22:0/1 OTE B9:0/6 EOR
%   B22:0/13  BFILT_BW  "UNIT B   FILTER BACKWASH" %
%   N34:49  "B VALVES AUTO/MANUAL CONTROL 0=AUTO 1=MANUAL" %
%   N34:91  "FILT B VALVE 13B CONTROL 0=AUTO 1=FORCE CLOSED 2=FORCE ON" %
%   B22:0/1  BFILT_OFFLINE  "B FORCED OFFLINE" %
%   B9:0/6  MV_013B  "ENERGIZE B BACKWASH INLET VALVE" %
% Rung: 15 %
SOR BST XIC B22:0/13 EQU N34:49 0 NXB EQU N34:49 1 EQU N34:25 2 BND XIO B22:0/1 OTE B9:0/8 EOR
%   B22:0/13  BFILT_BW  "UNIT B   FILTER BACKWASH" %
%   N34:49  "B VALVES AUTO/MANUAL CONTROL 0=AUTO 1=MANUAL" %
%   N34:25  "FILT B VALVE 14B CONTROL 0=AUTO 1=FORCE CLOSED 2=FORCE ON" %
%   B22:0/1  BFILT_OFFLINE  "B FORCED OFFLINE" %
%   B9:0/8  MV_014B  "ENERGIZE B BACKWASH OUTLET VALVE" %

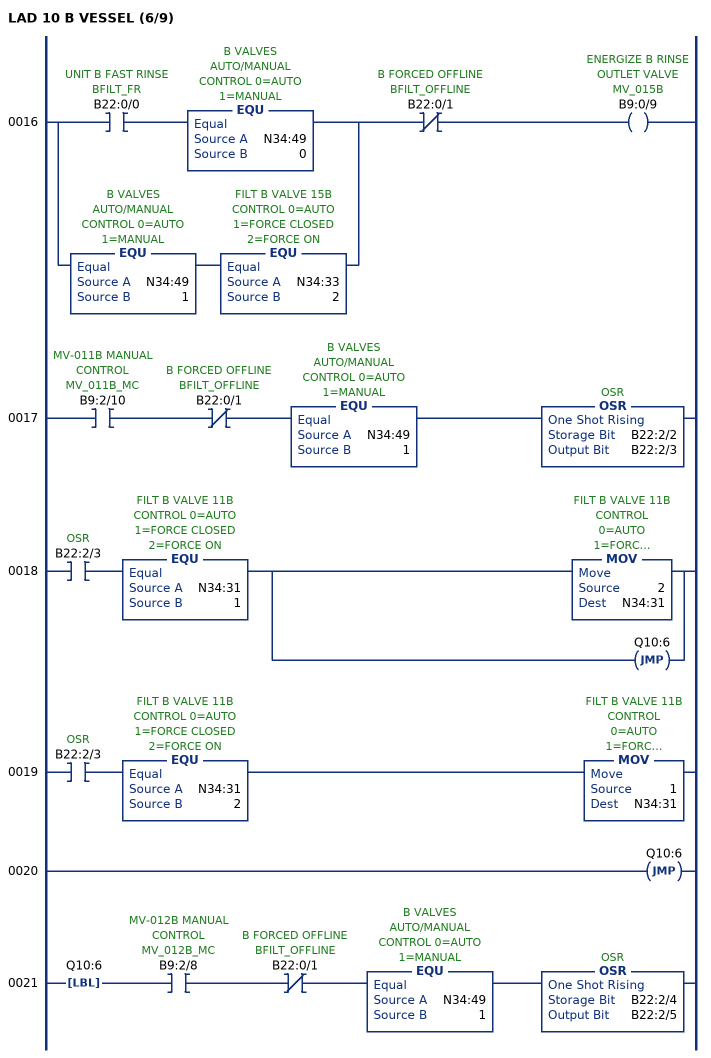
% Rung: 16 %
SOR BST XIC B22:0/0 EQU N34:49 0 NXB EQU N34:49 1 EQU N34:33 2 BND XIO B22:0/1 OTE B9:0/9 EOR
%   B22:0/0  BFILT_FR  "UNIT B FAST RINSE" %
%   N34:49  "B VALVES AUTO/MANUAL CONTROL 0=AUTO 1=MANUAL" %
%   N34:33  "FILT B VALVE 15B CONTROL 0=AUTO 1=FORCE CLOSED 2=FORCE ON" %
%   B22:0/1  BFILT_OFFLINE  "B FORCED OFFLINE" %
%   B9:0/9  MV_015B  "ENERGIZE B RINSE OUTLET VALVE" %
% Rung: 17 %
SOR XIC B9:2/10 XIO B22:0/1 EQU N34:49 1 OSR B22:2/2 B22:2/3 EOR
%   B9:2/10  MV_011B_MC  "MV-011B MANUAL CONTROL" %
%   B22:0/1  BFILT_OFFLINE  "B FORCED OFFLINE" %
%   N34:49  "B VALVES AUTO/MANUAL CONTROL 0=AUTO 1=MANUAL" %
%   B22:2/2  "OSR" %
%   B22:2/3  "OSR" %
% Rung: 18 %
SOR XIC B22:2/3 EQU N34:31 1 BST MOV 2 N34:31 NXB JMP Q10:6 BND EOR
%   B22:2/3  "OSR" %
%   N34:31  "FILT B VALVE 11B CONTROL 0=AUTO 1=FORCE CLOSED 2=FORCE ON" %
% Rung: 19 %
SOR XIC B22:2/3 EQU N34:31 2 MOV 1 N34:31 EOR
%   B22:2/3  "OSR" %
%   N34:31  "FILT B VALVE 11B CONTROL 0=AUTO 1=FORCE CLOSED 2=FORCE ON" %
% Rung: 20 %
SOR JMP Q10:6 EOR
% Rung: 21 %
SOR LBL Q10:6 XIC B9:2/8 XIO B22:0/1 EQU N34:49 1 OSR B22:2/4 B22:2/5 EOR
%   B9:2/8  MV_012B_MC  "MV-012B MANUAL CONTROL" %
%   B22:0/1  BFILT_OFFLINE  "B FORCED OFFLINE" %
%   N34:49  "B VALVES AUTO/MANUAL CONTROL 0=AUTO 1=MANUAL" %
%   B22:2/4  "OSR" %
%   B22:2/5  "OSR" %

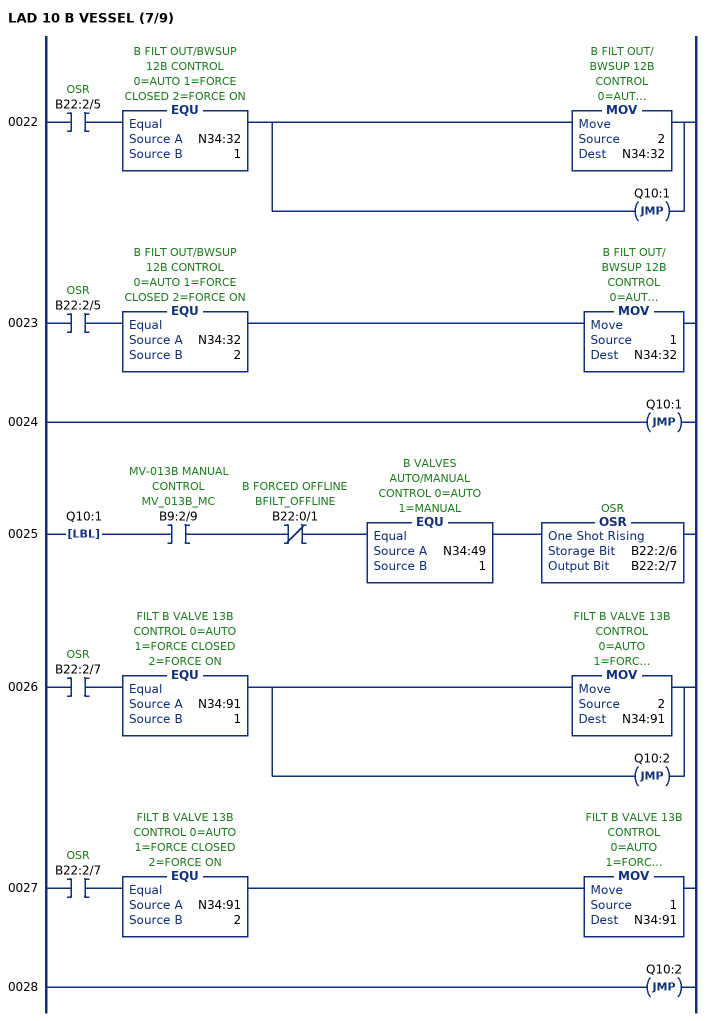
% Rung: 22 %
SOR XIC B22:2/5 EQU N34:32 1 BST MOV 2 N34:32 NXB JMP Q10:1 BND EOR
%   B22:2/5  "OSR" %
%   N34:32  "B FILT OUT/BWSUP 12B CONTROL 0=AUTO 1=FORCE CLOSED 2=FORCE ON" %
% Rung: 23 %
SOR XIC B22:2/5 EQU N34:32 2 MOV 1 N34:32 EOR
%   B22:2/5  "OSR" %
%   N34:32  "B FILT OUT/BWSUP 12B CONTROL 0=AUTO 1=FORCE CLOSED 2=FORCE ON" %
% Rung: 24 %
SOR JMP Q10:1 EOR
% Rung: 25 %
SOR LBL Q10:1 XIC B9:2/9 XIO B22:0/1 EQU N34:49 1 OSR B22:2/6 B22:2/7 EOR
%   B9:2/9  MV_013B_MC  "MV-013B MANUAL CONTROL" %
%   B22:0/1  BFILT_OFFLINE  "B FORCED OFFLINE" %
%   N34:49  "B VALVES AUTO/MANUAL CONTROL 0=AUTO 1=MANUAL" %
%   B22:2/6  "OSR" %
%   B22:2/7  "OSR" %
% Rung: 26 %
SOR XIC B22:2/7 EQU N34:91 1 BST MOV 2 N34:91 NXB JMP Q10:2 BND EOR
%   B22:2/7  "OSR" %
%   N34:91  "FILT B VALVE 13B CONTROL 0=AUTO 1=FORCE CLOSED 2=FORCE ON" %
% Rung: 27 %
SOR XIC B22:2/7 EQU N34:91 2 MOV 1 N34:91 EOR
%   B22:2/7  "OSR" %
%   N34:91  "FILT B VALVE 13B CONTROL 0=AUTO 1=FORCE CLOSED 2=FORCE ON" %
% Rung: 28 %
SOR JMP Q10:2 EOR

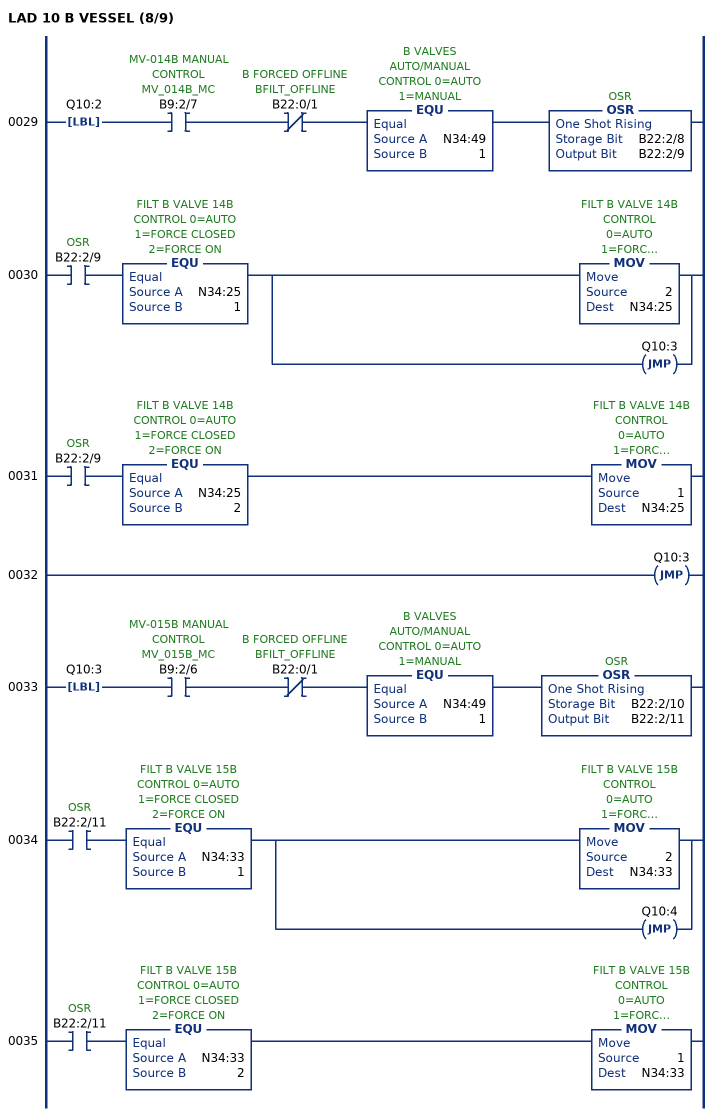
% Rung: 29 %
SOR LBL Q10:2 XIC B9:2/7 XIO B22:0/1 EQU N34:49 1 OSR B22:2/8 B22:2/9 EOR
%   B9:2/7  MV_014B_MC  "MV-014B MANUAL CONTROL" %
%   B22:0/1  BFILT_OFFLINE  "B FORCED OFFLINE" %
%   N34:49  "B VALVES AUTO/MANUAL CONTROL 0=AUTO 1=MANUAL" %
%   B22:2/8  "OSR" %
%   B22:2/9  "OSR" %
% Rung: 30 %
SOR XIC B22:2/9 EQU N34:25 1 BST MOV 2 N34:25 NXB JMP Q10:3 BND EOR
%   B22:2/9  "OSR" %
%   N34:25  "FILT B VALVE 14B CONTROL 0=AUTO 1=FORCE CLOSED 2=FORCE ON" %
% Rung: 31 %
SOR XIC B22:2/9 EQU N34:25 2 MOV 1 N34:25 EOR
%   B22:2/9  "OSR" %
%   N34:25  "FILT B VALVE 14B CONTROL 0=AUTO 1=FORCE CLOSED 2=FORCE ON" %
% Rung: 32 %
SOR JMP Q10:3 EOR
% Rung: 33 %
SOR LBL Q10:3 XIC B9:2/6 XIO B22:0/1 EQU N34:49 1 OSR B22:2/10 B22:2/11 EOR
%   B9:2/6  MV_015B_MC  "MV-015B MANUAL CONTROL" %
%   B22:0/1  BFILT_OFFLINE  "B FORCED OFFLINE" %
%   N34:49  "B VALVES AUTO/MANUAL CONTROL 0=AUTO 1=MANUAL" %
%   B22:2/10  "OSR" %
%   B22:2/11  "OSR" %
% Rung: 34 %
SOR XIC B22:2/11 EQU N34:33 1 BST MOV 2 N34:33 NXB JMP Q10:4 BND EOR
%   B22:2/11  "OSR" %
%   N34:33  "FILT B VALVE 15B CONTROL 0=AUTO 1=FORCE CLOSED 2=FORCE ON" %
% Rung: 35 %
SOR XIC B22:2/11 EQU N34:33 2 MOV 1 N34:33 EOR
%   B22:2/11  "OSR" %
%   N34:33  "FILT B VALVE 15B CONTROL 0=AUTO 1=FORCE CLOSED 2=FORCE ON" %

